Staubli VAL3: stopMove.pgx

public program stopMove()
begin
  stopMove()
end
